// TIA Portal V17 export
// export: Created 2025-03-07T09:19:50.5865384Z, ExportSetting WithDefaults, DisplayName Totally Integrated Automation Portal, DisplayVersion V17 Update 8, DisplayName TIA Portal Openness, DisplayVersion V17 Update 8, DisplayName TIA Portal Version Control Interface, DisplayVersion V17, DisplayName SINAMICS Startdrive Advanced, DisplayVersion V17 SP2, DisplayName SINAMICS Startdrive G110M, G120, G120C, G120D, G120P, G115D, DisplayVersion V17 SP2, DisplayName SINAMICS Startdrive G130, G150, S120, S150, SINAMICS MV, S210, DisplayVersion V17 SP2, DisplayName STEP 7 Professional, DisplayVersion V17 Update 8, DisplayName SINUMERIK ONE STEP 7 Toolbox, DisplayVersion V17 Update 12, DisplayName SINUMERIK 840D sl STEP 7 Toolbox, DisplayVersion V17 Update 12, DisplayName STEP 7 Safety, DisplayVersion V17 Update 6, DisplayName WinCC Advanced, DisplayVersion V17 Update 8
TYPE "SAFETY_BRAKE"
// stored: IsFailsafeCompliant false
   STRUCT
      GENERAL_CONDITIONS : Bool;   // GENERAL CONDITIONS
      BLOCK_CONDITIONS : Bool;   // BLOCK CONDITIONS
      UNBLOCK_CONDITIONS : Bool;   // UNBLOCK CONDITIONS
      GENERAL_CONDITIONS_HELP : Bool;   // GENERAL CONDITIONS HELP
      BLOCK_CONDITIONS_HELP : Bool;   // BLOCK CONDITIONS HELP
      UNBLOCK_CONDITIONS_HELP : Bool;   // UNBLOCK CONDITIONS HELP
      BLOCK_MANUAL_REQUEST : Bool;   // BLOCK MANUAL REQUEST
      UNBLOCK_MANUAL_REQUEST : Bool;   // UNBLOCK MANUAL REQUEST
      BLOCK_HMI_REQUEST : Bool;   // BLOCK HMI REQUEST
      UNBLOCK_HMI_REQUEST : Bool;   // UNBLOCK HMI REQUEST
      BLOCK_AUTO_REQUEST : Bool;   // BLOCK AUTO REQUEST
      UNBLOCK_AUTO_REQUEST : Bool;   // UNBLOCK AUTO REQUEST
      BLOCK_GLOBAL_REQUEST : Bool;   // BLOCK GLOBAL REQUEST
      UNBLOCK_GLOBAL_REQUEST : Bool;   // UNBLOCK GLOBAL REQUEST
      BLOCK_COMMAND : Bool;   // BLOCK COMMAND
      UNBLOCK_COMMAND : Bool;   // UNBLOCK COMMAND
      FULL_BLOCKED : Bool;   // BLOCK FEEDBACK / BLOCKED AND COMMANDED
      FULL_UNBLOCKED : Bool;   // UNBLOCK FEEDBACK / UNBLOCKED AND COMMANDED
      SIMULTANEITY_ALARM : Bool;   // SIMULTANEITY FAULT / SIMULTANEITY ALARM
      TIME_EXCEEDED_ALARM : Bool;   // TIME EXCEEDED / TIME EXCEEDED ALARM
      ANY_ACTIVE_ALARM : Bool;   // FAULT / ANY ACTIVE ALARM
      IS_SEOC_ALARMS : Bool;   // IMMEDIATE STOP AND STOP END OF CYCLE ALARMS
      PULSE_1 : Bool;   // PULSE 1
      PULSE_2 : Bool;   // PULSE 2
      PULSE_3 : Bool;   // PULSE 3
   END_STRUCT;
END_TYPE
